FUNCTION_BLOCK MultiReactors (* Composite Function Block Type *)
  (* Standard: 61499-2 *)
  (* Version 0.0, 9/17/2026, Schneider Electric, template *)
  PACKAGE SE.Nereda;
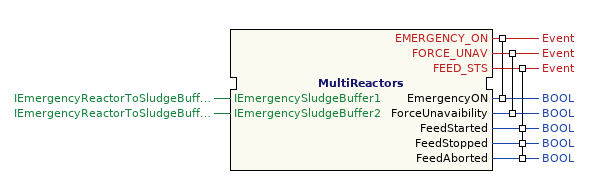
  EVENT_OUTPUT
    EMERGENCY_ON WITH EmergencyON;
    FORCE_UNAV WITH ForceUnavaibility;
    FEED_STS WITH FeedStarted, FeedStopped, FeedAborted;
  END_EVENT
  VAR_OUTPUT
    EmergencyON : BOOL;
    ForceUnavaibility : BOOL;
    FeedStarted : BOOL;
    FeedStopped : BOOL;
    FeedAborted : BOOL;
  END_VAR
  SOCKETS
    IEmergencySludgeBuffer1 : IEmergencyReactorToSludgeBuffer;
    IEmergencySludgeBuffer2 : IEmergencyReactorToSludgeBuffer;
  END_SOCKETS
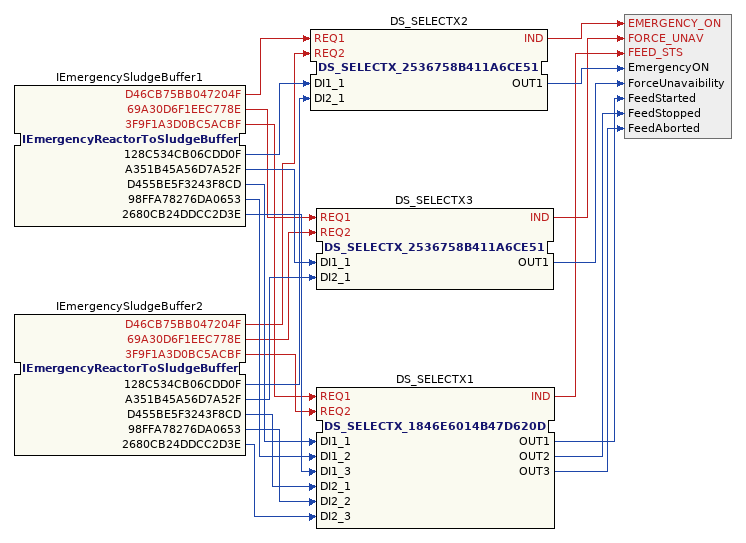
  FBS
    DS_SELECTX1 : DS_SELECTX_1846E6014B47D620D; {SET_ATTRIBUTE(Configuration.GenericFBType.InterfaceParams, Runtime.Standard#CNTX:=2;CNTY:=3;DI${CNTX,_,CNTY$}:BOOL,BOOL,BOOL)} {SET_ATTRIBUTE(Configuration.Component.HideUnusedPorts, )}
    DS_SELECTX2 : DS_SELECTX_2536758B411A6CE51; {SET_ATTRIBUTE(Configuration.GenericFBType.InterfaceParams, Runtime.Standard#CNTX:=2;CNTY:=1;DI${CNTX,_,CNTY$}:BOOL)} {SET_ATTRIBUTE(Configuration.Component.HideUnusedPorts, )}
    DS_SELECTX3 : DS_SELECTX_2536758B411A6CE51; {SET_ATTRIBUTE(Configuration.GenericFBType.InterfaceParams, Runtime.Standard#CNTX:=2;CNTY:=1;DI${CNTX,_,CNTY$}:BOOL)} {SET_ATTRIBUTE(Configuration.Component.HideUnusedPorts, )}
  END_FBS
  EVENT_CONNECTIONS
    IEmergencySludgeBuffer1.D46CB75BB047204F TO DS_SELECTX2.REQ1;
    IEmergencySludgeBuffer1.69A30D6F1EEC778E TO DS_SELECTX3.REQ1;
    IEmergencySludgeBuffer1.3F9F1A3D0BC5ACBF TO DS_SELECTX1.REQ1;
    IEmergencySludgeBuffer2.D46CB75BB047204F TO DS_SELECTX2.REQ2;
    IEmergencySludgeBuffer2.69A30D6F1EEC778E TO DS_SELECTX3.REQ2;
    IEmergencySludgeBuffer2.3F9F1A3D0BC5ACBF TO DS_SELECTX1.REQ2;
    DS_SELECTX2.IND TO EMERGENCY_ON;
    DS_SELECTX3.IND TO FORCE_UNAV;
    DS_SELECTX1.IND TO FEED_STS;
  END_CONNECTIONS
  DATA_CONNECTIONS
    IEmergencySludgeBuffer1.128C534CB06CDD0F TO DS_SELECTX2.DI1_1;
    IEmergencySludgeBuffer1.A351B45A56D7A52F TO DS_SELECTX3.DI1_1;
    IEmergencySludgeBuffer1.D455BE5F3243F8CD TO DS_SELECTX1.DI1_1;
    IEmergencySludgeBuffer1.98FFA78276DA0653 TO DS_SELECTX1.DI1_2;
    IEmergencySludgeBuffer1.2680CB24DDCC2D3E TO DS_SELECTX1.DI1_3;
    IEmergencySludgeBuffer2.128C534CB06CDD0F TO DS_SELECTX2.DI2_1;
    IEmergencySludgeBuffer2.A351B45A56D7A52F TO DS_SELECTX3.DI2_1;
    IEmergencySludgeBuffer2.D455BE5F3243F8CD TO DS_SELECTX1.DI2_1;
    IEmergencySludgeBuffer2.98FFA78276DA0653 TO DS_SELECTX1.DI2_2;
    IEmergencySludgeBuffer2.2680CB24DDCC2D3E TO DS_SELECTX1.DI2_3;
    DS_SELECTX2.OUT1 TO EmergencyON;
    DS_SELECTX3.OUT1 TO ForceUnavaibility;
    DS_SELECTX1.OUT1 TO FeedStarted;
    DS_SELECTX1.OUT2 TO FeedStopped;
    DS_SELECTX1.OUT3 TO FeedAborted;
  END_CONNECTIONS
END_FUNCTION_BLOCK
